// Mitsubishi GX Works2 project: z01   PLC: Q02/Q02H

PROGRAM MAIN
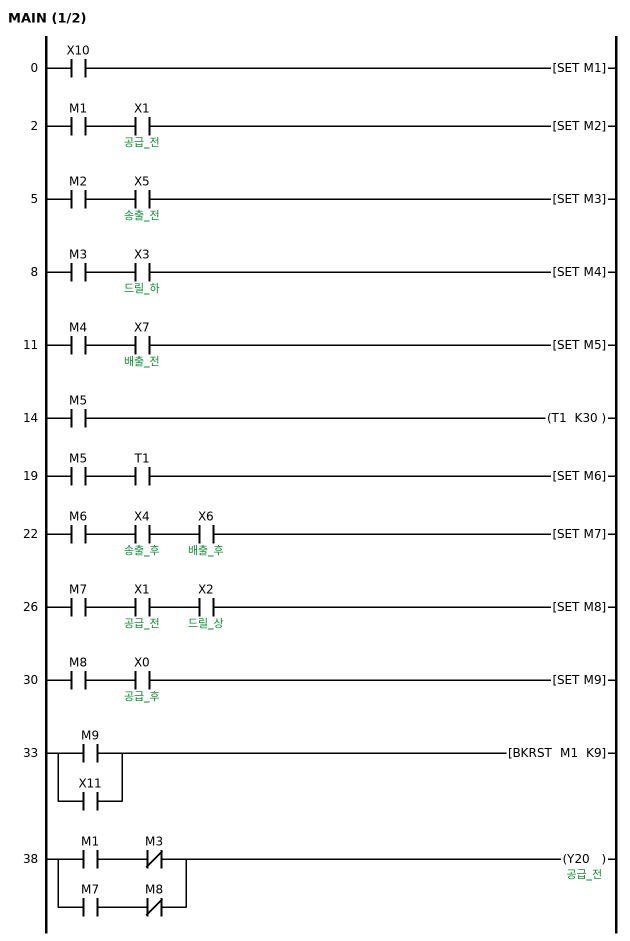
0     LD      X10
      SET     M1
2     LD      M1
      AND     X1  ; 공급_전
      SET     M2
5     LD      M2
      AND     X5  ; 송출_전
      SET     M3
8     LD      M3
      AND     X3  ; 드릴_하
      SET     M4
11    LD      M4
      AND     X7  ; 배출_전
      SET     M5
14    LD      M5
      OUT     T1 K30
19    LD      M5
      AND     T1
      SET     M6
22    LD      M6
      AND     X4  ; 송출_후
      AND     X6  ; 배출_후
      SET     M7
26    LD      M7
      AND     X1  ; 공급_전
      AND     X2  ; 드릴_상
      SET     M8
30    LD      M8
      AND     X0  ; 공급_후
      SET     M9
33    LD      M9
      OR      X11
      BKRST   M1 K9
38    LD      M1
      ANI     M3
      LD      M7
      ANI     M8
      ORB
      OUT     Y20  ; 공급_전
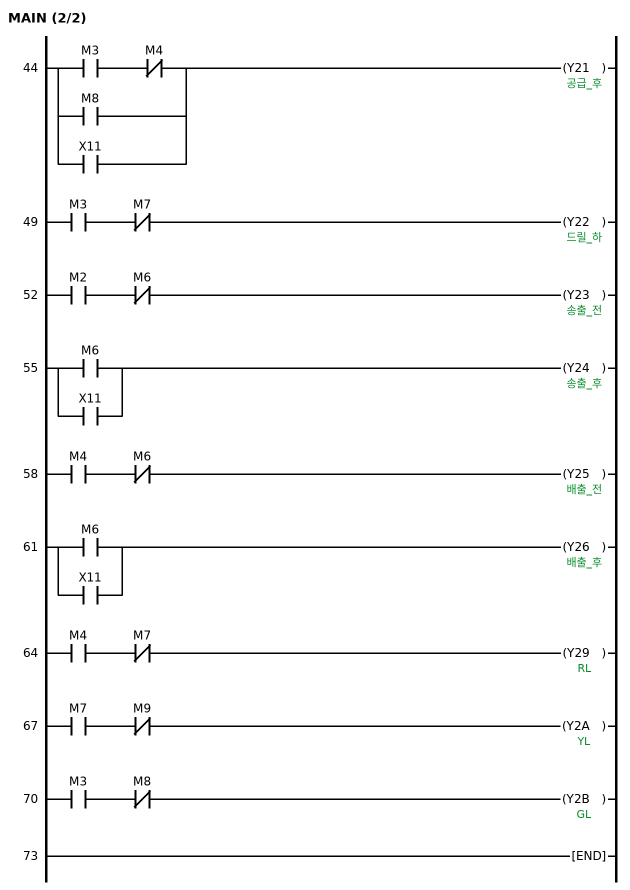
44    LD      M3
      ANI     M4
      OR      M8
      OR      X11
      OUT     Y21  ; 공급_후
49    LD      M3
      ANI     M7
      OUT     Y22  ; 드릴_하
52    LD      M2
      ANI     M6
      OUT     Y23  ; 송출_전
55    LD      M6
      OR      X11
      OUT     Y24  ; 송출_후
58    LD      M4
      ANI     M6
      OUT     Y25  ; 배출_전
61    LD      M6
      OR      X11
      OUT     Y26  ; 배출_후
64    LD      M4
      ANI     M7
      OUT     Y29  ; RL
67    LD      M7
      ANI     M9
      OUT     Y2A  ; YL
70    LD      M3
      ANI     M8
      OUT     Y2B  ; GL
73    END
END_PROGRAM
